INTERFACE I_HE_SATT_Commands


PROPERTY PermitMove : BOOL
GET
END_GET
END_PROPERTY


PROPERTY Reset : BOOL
GET
END_GET
END_PROPERTY

END_INTERFACE

(* stored: Version 1.1.0.1
   Itf I_HE_SATT_Commands: Id {a08734bf-785c-4688-8c5d-7461eb32ca94}
   Property PermitMove: Id {6e4d309d-0b60-41ee-a05a-62ef3d3fa462}
   Get Get: Id {bb4137e3-a65c-492e-85c6-fd552e96faf4}
   Property Reset: Id {3270352f-256d-4cb6-9760-b157566f6f50}
   Get Get: Id {3feb3014-39d2-4a7c-9b15-892de56959b9} *)
